FUNCTION_BLOCK RealValueChanged (* Basic Function Block Type *)
  (* Standard: 61499-2 *)
  (* Version 0.0, 6/25/2026, Schneider Electric, Template *)
  PACKAGE SE.Nereda;
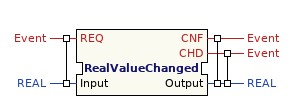
  EVENT_INPUT
    REQ WITH Input; (* Normal Execution Request *)
  END_EVENT
  EVENT_OUTPUT
    CNF WITH Output; (* Execution Confirmation *)
    CHD WITH Output;
  END_EVENT
  VAR_INPUT
    Input : REAL; (* Input event qualifier *)
  END_VAR
  VAR_OUTPUT
    Output : REAL; (* Output event qualifier *)
  END_VAR
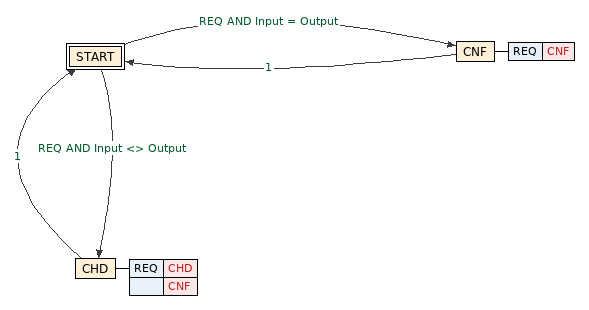
  EC_STATES
    START; (* Initial State *)
    CNF : REQ -> CNF;
    CHD : REQ -> CHD, -> CNF;
  END_STATES
  EC_TRANSITIONS
    CHD TO START := 1;
    CNF TO START := 1;
    START TO CHD := REQ AND Input <> Output;
    START TO CNF := REQ AND Input = Output;
  END_TRANSITIONS
  ALGORITHM REQ IN ST: (* Normally executed algorithm *)
;
Output := Input;
  END_ALGORITHM
END_FUNCTION_BLOCK
